// TIA Portal V16 export
// export: Created 2021-11-12T13:31:05.4485671Z, ExportSetting WithDefaults, DisplayName Totally Integrated Automation Portal, DisplayVersion V16 Update 3, DisplayName TIA Portal Version Control Interface, DisplayVersion V16 Update 2, DisplayName TIA Portal Openness, DisplayVersion V16 Update 3, DisplayName SINAMICS Startdrive Advanced, DisplayVersion V16 Update 5, DisplayName SINAMICS Startdrive G130, G150, S120, S150, SINAMICS MV, S210, DisplayVersion V16 Update 5, DisplayName SINAMICS Startdrive G110M, G120, G120C, G120D, G120P, G115D, DisplayVersion V16 Update 5, DisplayName STEP 7 Professional, DisplayVersion V16 Update 3, DisplayName STEP 7 Safety, DisplayVersion V16, DisplayName WinCC UA Professional, DisplayVersion V16 Update 3
DATA_BLOCK "ProdParam"   // DB3
{ S7_Optimized_Access := 'TRUE'; DB_Accessible_From_OPC_UA := 'FALSE' }
VERSION : 0.1
// stored: AutoNumber true, DBAccessibleFromOPCUA false, IsOnlyStoredInLoadMemory false, IsRetainMemResEnabled false, IsWriteProtectedInAS false, MemoryReserve 100
   VAR RETAIN
      PartType : Int := 2163;   // Production type
      DayNumber : Int := 0;   // Pořadové číslo dne
      Melt : String[3] := 'B5';   // Tavba
      KAS1_RodDiam : Int := 0;   // KAS1 - rod diameter
      KAS1_RodLength : Int := 0;   // KAS1 - rod length
      KAS1_PartLength : Int := 450;   // KAS1 - part length
      KAS2_RodDiam : Int := 0;   // KAS2 - rod diameter
      KAS2_RodLength : Int := 0;   // KAS2 - rod length
      KAS2_PartLength : Int := 450;   // KAS2 - part length
      "110_ConvSpeed" : Real := 1200.0;   // 110 - Conveyor speed
      "110_ConvSpeedSlow" : Real := 400.0;   // 110 - Conveyor speed slow
      "120_ConvSpeed" : Real := 1200.0;   // 120 - Conveyor speed
      "120_ConvSpeedSlow" : Real := 400.0;   // 120 - Conveyor speed slow
      BSN1_MinTime : Real := 0.0;   // BSN1 - minimum heating time
      BSN1_MaxTime : Real := 0.0;   // BSN1 - maximum heating time
      BSN1_StepTime : Real := 71.0;   // BSN1 - time to next step [s]
      BSN1_StepLength : Int := 2;   // BSN1 - length of step [mm]
      BSN1_TempZone1 : Real := 5301.0;   // BSN1 - setpoint temperature zone 1
      BSN1_TempZone2 : Real := 5301.0;   // BSN1 - setpoint temperature zone 2
      BSN1_TempZone3 : Real := 5501.0;   // BSN1 - setpoint temperature zone 3
      BSN1_TempZone4 : Real := 5501.0;   // BSN1 - setpoint temperature zone 4
      BSN1_TempZone5 : Real := 5501.0;   // BSN1 - setpoint temperature zone 5
      BSN1_NrOfLines : Int := 4;   // BSN1 - number of used lines in map
      BSN2_StepTime : Real := 70.0;   // BSN2 - time to next step [s]
      BSN2_StepLength : Int := 2;   // BSN2 - length of step [mm]
      BSN2_MinTime : Real := 0.0;   // BSN2 - minimum heating time
      BSN2_MaxTime : Real := 0.0;   // BSN2 - maximum heating time
      BSN2_TempZone1 : Real := 5300.0;   // BSN2 - setpoint temperature zone 1
      BSN2_TempZone2 : Real := 5302.0;   // BSN2 - setpoint temperature zone 2
      BSN2_TempZone3 : Real := 5502.0;   // BSN2 - setpoint temperature zone 3
      BSN2_TempZone4 : Real := 5502.0;   // BSN2 - setpoint temperature zone 4
      BSN2_TempZone5 : Real := 5502.0;   // BSN2 - setpoint temperature zone 5
      BSN2_NrOfLines : Int := 4;   // BSN2 - number of used lines in map
      "210_BoxWrn" : Int := 0;   // 210 - Number of part in box when warning occurs
      "210_BoxErr" : Int := 0;   // 210 - Number of part in box when error occurs
      "210_ConvSpeed" : Real := 1000.0;   // 210 - Conveyor speed
      "210_ConvSpeedSlow" : Real := 460.0;   // 210 - Conveyor speed slow
      "220_BoxWrn" : Int := 0;   // 220 - Number of part in box when warning occurs
      "220_BoxErr" : Int := 0;   // 220 - Number of part in box when error occurs
      "220_ConvSpeed" : Real := 1000.0;   // 220 - Conveyor speed
      "220_ConvSpeedSlow" : Real := 460.0;   // 220 - Conveyor speed slow
      "230_BoxWrn" : Int := 0;   // 230 - Number of part in box when warning occurs
      "230_BoxErr" : Int := 0;   // 230 - Number of part in box when error occurs
      "230_GL01_ConvSpeed" : Real := 1000.0;   // 230 - Conveyor speed
      "230_GL01_ConvSpeedSlow" : Real := 460.0;   // 220 - Conveyor speed slow
      "230_GL02_ConvSpeed" : Real := 1000.0;   // 230 - Conveyor speed
      "230_GL02_ConvSpeedSlow" : Real := 460.0;   // 220 - Conveyor speed slow
      MaxTime_BSN1_SCH1 : Int := 0;   // Maximum time from BSN1 to SCH1
      MaxTime_BSN1_SCH1Die3 : Int := 0;   // Maximum time from furnace to press in die 3
      MaxTime_BSN1_SCH1Die4 : Int := 0;   // Maximum time from furnace to press in die 4
      MaxTime_BSN1_SCH1Die5 : Int := 0;   // Maximum time from furnace to press in die 5
      MaxTime_BSN1_SCH1Die6 : Int := 0;   // Maximum time from furnace to press in die 6
      MaxTime_BSN1_SCH1Die7 : Int := 0;   // Maximum time from furnace to cut in die 7
      MaxTime_BSN1_BSN3 : Int := 0;   // Maximum time from BSN1 to BSN3
      "2R1_LubeAmount1" : UInt := 0;   // amount of material 1 diluted in water
      "2R1_LubeAmount2" : UInt := 0;   // amount of material 1 diluted in water
      "2R1_WaterAmount" : UInt := 0;   // amount of water for dilution
      SCH1_TempUpper1 : Int := 1;   // SCH1 - Temperature setpoint for upper tool
      SCH1_TempLower1 : Int := 1;   // SCH1 - Temperature setpoint for lower tool
      SCH1_TempUpper2 : Int := 1;   // SCH1 - Temperature setpoint for upper tool
      SCH1_TempLower2 : Int := 1;   // SCH1 - Temperature setpoint for lower tool
      SCH1_TempTolerance : Int := 20;   // SCH1 - Tolerance of temperature of tool
      BSN3_MinTime : Real := 0.0;   // BSN3 - minimum heating time
      BSN3_MaxTime : Real := 0.0;   // BSN3 - maximum heating time
      BSN3_TempZone1 : Real := 5000.0;   // BSN3 - setpoint temperature zone 1
      BSN3_TempZone2 : Real := 5101.0;   // BSN3 - setpoint temperature zone 2
      BSN3_TempZone3 : Real := 5101.0;   // BSN3 - setpoint temperature zone 3
      BSN3_TempZone4 : Real := 5101.0;   // BSN3 - setpoint temperature zone 4
      BSN3_TempZone5 : Real := 5101.0;   // BSN3 - setpoint temperature zone 5
      BSN3_TempZone6 : Real := 5101.0;   // BSN3 - setpoint temperature zone 6
      BSN3_TempZone7 : Real := 5005.0;   // BSN3 - setpoint temperature zone 7
      BSN3_ActPartTime : Real := 1.0;   // BSN3 - actual setpoint of time in furnace according to belt speed [min]
      BSN3_BoxWrn : Int := 0;   // BSN3 - Number of part in box when warning occurs
      BSN3_BoxErr : Int := 0;   // BSN3 - Number of part in box when error occurs
      "310_Temp" : Real := 40.0;   // 310 - setpoint temperature
      "310_TempHys" : Real := 5.0;   // 310 - temperature hysteresys
      "320_ConvSpeed" : Real := 700.0;   // 320 - Conveyor speed
      "320_ConvSpeedSlow" : Real := 460.0;   // 320 - Conveyor speed slow
      "330_BoxWrn" : Int := 0;   // 330 - Number of part in box when warning occurs
      "330_BoxErr" : Int := 0;   // 330 - Number of part in box when error occurs
      "330_GL01_ConvSpeed" : Real := 400.0;   // 330 - Conveyor speed
      "330_GL01_ConvSpeedSlow" : Real := 200.0;   // 320 - Conveyor speed slow
      "330_GL02_ConvSpeed" : Real := 400.0;   // 330 - Conveyor speed
      "330_GL02_ConvSpeedSlow" : Real := 200.0;   // 320 - Conveyor speed slow
      "330_GL03_ConvSpeed" : Real := 400.0;   // 330 - Conveyor speed
      "330_GL03_ConvSpeedSlow" : Real := 200.0;   // 320 - Conveyor speed slow
      BSN4_MinTime : Real := 0.0;   // BSN4 - minimum heating time
      BSN4_MaxTime : Real := 0.0;   // BSN4 - maximum heating time
      BSN4_TempZone1 : Real := 5004.0;   // BSN4 - setpoint temperature zone 1
      BSN4_TempZone2 : Real := 5004.0;   // BSN4 - setpoint temperature zone 2
      BSN4_TempZone3 : Real := 5004.0;   // BSN4 - setpoint temperature zone 3
      BSN4_TempZone4 : Real := 5004.0;   // BSN4 - setpoint temperature zone 4
      BSN4_TempZone5 : Real := 5004.0;   // BSN4 - setpoint temperature zone 5
      BSN4_TempZone6 : Real := 5004.0;   // BSN4 - setpoint temperature zone 6
      BSN4_TempZone7 : Real := 5004.0;   // BSN4 - setpoint temperature zone 7
      BSN4_ActPartTime : Real := 2.0;   // BSN4 - actual setpoint of time in furnace according to belt speed [min]
      "410_Temp" : Real := 40.0;   // 410 - setpoint temperature
      "410_TempHys" : Real := 5.0;   // 410 - temperature hysteresys
      "430_ConvSpeed" : Real := 700.0;   // 430 - Conveyor speed
      "430_ConvSpeedSlow" : Real := 1400.0;   // 430 - Conveyor speed slow
      "450_BoxWrn" : Int := 0;   // 450 - Number of part in box when warning occurs
      "450_BoxErr" : Int := 0;   // 450 - Number of part in box when error occurs
      "450_GL01_ConvSpeed" : Real := 400.0;   // 450 - Conveyor speed
      "450_GL01_ConvSpeedSlow" : Real := 200.0;   // 450 - Conveyor speed slow
      "450_GL02_ConvSpeed" : Real := 400.0;   // 450 - Conveyor speed
      "450_GL02_ConvSpeedSlow" : Real := 200.0;   // 450 - Conveyor speed slow
      "450_GL03_ConvSpeed" : Real := 400.0;   // 450 - Conveyor speed
      "450_GL03_ConvSpeedSlow" : Real := 200.0;   // 450 - Conveyor speed slow
      "450_GL04_ConvSpeed" : Real := 400.0;   // 450 - Conveyor speed
      "450_GL04_ConvSpeedSlow" : Real := 200.0;   // 450 - Conveyor speed slow
      BSN5_MinTime : Real := 0.0;   // BSN5 - minimum heating time
      BSN5_MaxTime : Real := 0.0;   // BSN5 - maximum heating time
      BSN5_TempZone1 : Real := 0.0;   // BSN5 - setpoint temperature zone 1
      BSN5_TempZone2 : Real := 0.0;   // BSN5 - setpoint temperature zone 2
      BSN5_TempZone3 : Real := 0.0;   // BSN5 - setpoint temperature zone 3
      BSN5_TempZone4 : Real := 0.0;   // BSN5 - setpoint temperature zone 4
      BSN5_TempZone5 : Real := 0.0;   // BSN5 - setpoint temperature zone 5
      BSN5_TempZone6 : Real := 0.0;   // BSN5 - setpoint temperature zone 6
      BSN5_TempZone7 : Real := 0.0;   // BSN5 - setpoint temperature zone 7
      BSN5_ActPartTime : Real := 0.0;   // BSN5 - actual setpoint of time in furnace according to belt speed [min]
      "420_Temp" : Real := 40.0;   // 420 - setpoint temperature
      "420_TempHys" : Real := 5.0;   // 420 - temperature hysteresys
      "440_ConvSpeed" : Real := 700.0;   // 440 - Conveyor speed
      "440_ConvSpeedSlow" : Real := 1400.0;   // 440 - Conveyor speed slow
      "460_BoxWrn" : Int := 0;   // 460 - Number of part in box when warning occurs
      "460_BoxErr" : Int := 0;   // 460 - Number of part in box when error occurs
      "460_GL01_ConvSpeed" : Real := 400.0;   // 460 - Conveyor speed
      "460_GL01_ConvSpeedSlow" : Real := 200.0;   // 460 - Conveyor speed slow
      "460_GL02_ConvSpeed" : Real := 400.0;   // 460 - Conveyor speed
      "460_GL02_ConvSpeedSlow" : Real := 200.0;   // 460 - Conveyor speed slow
      "460_GL03_ConvSpeed" : Real := 400.0;   // 460 - Conveyor speed
      "460_GL03_ConvSpeedSlow" : Real := 200.0;   // 460 - Conveyor speed slow
      "460_GL04_ConvSpeed" : Real := 400.0;   // 460 - Conveyor speed
      "460_GL04_ConvSpeedSlow" : Real := 200.0;   // 460 - Conveyor speed slow
   END_VAR
BEGIN
END_DATA_BLOCK
